ABB RAPID module: HSLU_Data.modx

MODULE HSLU_Data

    !************************************************
    ! Declaration :     string
    !************************************************
    !
    TASK PERS string st_HSLU_Header:="Swissbau";

    !************************************************
    ! Declaration :     num
    !************************************************
    !
    TASK PERS num n_HSLU_ActOverride:=0;

ENDMODULE
